Fanuc KAREL source: ko00130.KL

PROGRAM KO00130
%STACKSIZE=65535
%PRIORITY=65535
%NOLOCKGROUP
VAR
R : REAL
OUT : XYZWPR
N : REAL
-- UNRESOLVED DECLARATIONS (source type spelling not recovered)
-- CFG : TYPE_0x001C (type_u16=0x001C)
BEGIN
N=1
R=2.0
-- UNRESOLVED_PC line 11 opcodes [9D 22 A5] marker_code=29
-- UNRESOLVED_PC line 12 opcodes [27 22 22 22 22 22 22 22 76 7E 4A] marker_code=44
END KO00130
